ABB RAPID module: CalibData.modx

MODULE CalibData
    PERS tooldata CONST_EE_TOOL_EGP_C_40 := [TRUE,[[0.0, 0.0, 124.1], [1.0, 0.0, 0.0 , 0.0] ], [0.62, [5.3, -0.009, 43.66], [1.0, 0.0, 0.0, 0.0], 0.0, 0.0, 0.0]];
ENDMODULE
